(*********************************** G.D S.p.A. - Technical Department ***********************************
============= PROGRAM INFO ============
FOLDER:             TBD
MACHINES INVOLVED:  TBD 

============= DESCRIPTION =============
csp machine declaration

============= REVISIONS ===============
Date		Version	 	Author      	Description             
----------	-------		------------  	--------------------------------------------
2019/04/05 	0000.00	 	M.Grasso		Creation of the PRG
2020/05/05 	0000.01	 	G.Imbriaco		From original author, G.Imbriaco: AccU Change motor with absolute encoder and brake.
										If position_req_mm parameter different from actual_pos_mm and machine reset_edge
										the motor move to position_req then disable again
										Manual movement with basc axis object under test( preset, moving,...)
										All disabled if main accU_Change is not Operational

**********************************************************************************************************)
(*$R process_ref := prc; $*)
PROGRAM csp_case_transport_accU_depth
VAR
	
	prc:											process;
	prc_path:										STRING;
	
	axis:											axis;
	Slot24_drv:										coe_drive;

	not_in_position:								message;
	axis_restore_absolute_position_fb:				restore_absolute_position_with_retain_fb;

	disable_req:									BOOL:=FALSE;
	position_req_mm:								LREAL:=0.0;(*$P unit:= mm; $*)
	move_velocity_req_mms:							LREAL:=10.0;(*$P unit:= mm; $*)
	position_req_tolerance_mm:						LREAL:=0.2;	(*$P $*)
	
	axis_status:									axis_status_enum := AXIS_STATUS_PARAMETERS_START;(*$M $*)
	in_position:									BOOL:=FALSE;(*$M $*)	
	actual_position_mm:								LREAL:=0.0; (*$M unit:= mm; $*)
	axis_move_condition:							BOOL:=FALSE;
	torque_limit:                                   INT := 5000;    (*$P $*)
    torque_limit_old:                               INT;
	
	in_position_motcond:							motorization_conditioner;
	fsm_status:										csp_case_transport_accU_depth_enum;(*$M $*)
	fsm_next_status:								csp_case_transport_accU_depth_enum;
	fsm_enable_condition:							BOOL:=FALSE;
	debug_state_machine:							BOOL:=FALSE;
	debug_state_machine_one_step:					BOOL:=FALSE;
	NC_encoder_val AT %I*:							DINT;
	
END_VAR
VAR PERSISTENT
	per_encoder_val:								UDINT;
	axis_restore_absolute_position_data:			restore_absolute_position_with_retain_struct;
END_VAR

_read_var_input();

_object_manager();

IF NOT objects_running()
THEN
	RETURN;	
END_IF

_read_process_image();

_mode_manager();

CASE process_get_mode(prc) OF
	MODE_ABSENT,
	MODE_INACTIVE:
		RETURN;
	MODE_TEST:
		_handle_process_test();
END_CASE

_set_runtime_properties();

(********************************* BODY *********************************)
//Axis Torque Limit
IF torque_limit <> Torque_limit_old
    THEN
    IF coe_drive_write_parameter(
        index:=16#7010 ,
        complete_access:= FALSE ,
        sub_index:= 16#0B,
        data_source:= ADR(torque_limit),
        data_lenght:= SIZEOF(torque_limit),
        CONVERSION_this:=csp_case_transport_accU_depth.axis.coe_drive^ )= COE_DRIVE_RETURN_VALUE_DONE
       THEN
		 torque_limit_old := Torque_limit;
	END_IF
END_IF

//Axis move condition
IF 	csp_main_accuChange.case_transport_accU_depth_move_req
	OR jog_manager_is_jog_axis_active(SMTR61210_SMTR61200_SMTR61420_CASE_FEED_SHUTTLE_TRANSPORT_AND_DISCHARGE_DEPTH, csp_main_jogManager.jog_manager_accuchange)
THEN
	axis_move_condition := TRUE;
ELSE
	axis_move_condition := FALSE;
END_IF

(*FSM Control*)
fsm_enable_condition := axis_is_ok(FALSE, axis)
						AND
						process_subtree_is_ready(prc)
						AND
						process_get_mode(csp_main_accuChange.prc) = MODE_OPERATIONAL
						AND
						axis_restore_absolute_position_fb.o_position_restored
						AND
						NOT disable_req;		
					
IF	(NOT fsm_enable_condition
	OR
	disable_req)
	AND
	fsm_status <> CSP_CASE_TRANSPORT_ACCU_DEPTH_STATUS_DISABLED
	AND
	fsm_status < CSP_CASE_TRANSPORT_ACCU_DEPTH_STATUS_STOP_REQUEST
THEN
	fsm_status	:=	CSP_CASE_TRANSPORT_ACCU_DEPTH_STATUS_STOP_REQUEST;
END_IF

CASE fsm_status OF
	
	CSP_CASE_TRANSPORT_ACCU_DEPTH_STATUS_NOT_INITIALIZED:
	
        IF	axis_is_ok(return_when_absent := TRUE, CONVERSION_this := axis)
        THEN
            fsm_next_status := CSP_CASE_TRANSPORT_ACCU_DEPTH_STATUS_DISABLED;
        END_IF

		
	CSP_CASE_TRANSPORT_ACCU_DEPTH_STATUS_DISABLED:
	
		IF	fsm_enable_condition
		THEN
			(* Axis with absolute encoder, no home procedure request *)
			fsm_next_status := CSP_CASE_TRANSPORT_ACCU_DEPTH_STATUS_POSITION_CHECK;
		END_IF;
	
		
	CSP_CASE_TRANSPORT_ACCU_DEPTH_STATUS_POSITION_CHECK:

		IF 	axis_move_condition
			OR jog_manager_is_jog_axis_active(SMTR61210_SMTR61200_SMTR61420_CASE_FEED_SHUTTLE_TRANSPORT_AND_DISCHARGE_DEPTH, csp_main_jogManager.jog_manager_accuchange)
		THEN
			fsm_next_status := CSP_CASE_TRANSPORT_ACCU_DEPTH_STATUS_ENABLE_REQUEST;
		END_IF			
	
		
	CSP_CASE_TRANSPORT_ACCU_DEPTH_STATUS_ENABLE_REQUEST:
	
		axis_enable(axis);
		IF axis_is_standstill(axis)
		THEN
			fsm_next_status	:=	CSP_CASE_TRANSPORT_ACCU_DEPTH_STATUS_ENABLED;
		END_IF		

		
	CSP_CASE_TRANSPORT_ACCU_DEPTH_STATUS_ENABLED:
	
		IF 	axis_move_condition
			OR jog_manager_is_jog_axis_active(SMTR61210_SMTR61200_SMTR61420_CASE_FEED_SHUTTLE_TRANSPORT_AND_DISCHARGE_DEPTH, csp_main_jogManager.jog_manager_accuchange)
		THEN
			fsm_next_status	:= CSP_CASE_TRANSPORT_ACCU_DEPTH_STATUS_PHASE_TO_MASTER;	
		END_IF
		
		
	CSP_CASE_TRANSPORT_ACCU_DEPTH_STATUS_PHASE_TO_MASTER:

		IF 	axis.actual_position <> csp_case_transport_accu_virtualMaster.axis.actual_position
			AND ABS(axis.actual_position - csp_case_transport_accu_virtualMaster.axis.actual_position) < 5
		THEN
			axis_move_absolute(
				position 		:= csp_case_transport_accu_virtualMaster.axis.actual_position,
				velocity 		:= move_velocity_req_mms,
				direction		:= AXIS_SHORTEST_WAY,
				acceleration 	:= csp_main_accuChange.CONSTANTS.MAX_ACCELERATION_MMpSEC2 * 0.1,
				deceleration 	:= csp_main_accuChange.CONSTANTS.MAX_DECELERATION_MMpSEC2 * 0.1,
				jerk 			:= csp_main_accuChange.CONSTANTS.MAX_JERK_MMpSEC3, 
				buffer_mode 	:= AXIS_BUFFER_MODE_BUFFERED,
				CONVERSION_this := axis
				); 	
		END_IF
		
		IF 	axis_is_absolute_moving(axis)
			OR axis.actual_position = csp_case_transport_accu_virtualMaster.axis.actual_position
		THEN
			fsm_next_status	:= CSP_CASE_FEED_SHUTTLE_ACCU_DEPTH_STATUS_GEAR_REQUEST;
		END_IF
			
		
	CSP_CASE_TRANSPORT_ACCU_DEPTH_STATUS_GEAR_REQUEST:

		IF	axis_is_standstill(axis)
			AND (
					csp_case_transport_accU_virtualMaster.master_redefined
					OR jog_manager_is_jog_axis_active(SMTR61210_SMTR61200_SMTR61420_CASE_FEED_SHUTTLE_TRANSPORT_AND_DISCHARGE_DEPTH, csp_main_jogManager.jog_manager_accuchange)
				)
		THEN
			axis_engage_position_gear(
				ratio 			:= 1.0,
				acceleration 	:= csp_main_accuChange.CONSTANTS.MAX_ACCELERATION_MMpSEC2 * 0.1,
				deceleration 	:= csp_main_accuChange.CONSTANTS.MAX_DECELERATION_MMpSEC2 * 0.1,
				jerk			:= csp_main_accuChange.CONSTANTS.MAX_JERK_MMpSEC3,
				master 			:= csp_case_transport_accU_virtualMaster.axis,
				CONVERSION_this := axis);
			
		END_IF
		
		IF axis_is_gear_engaging(axis)
		THEN
			fsm_next_status	:=	CSP_CASE_TRANSPORT_ACCU_DEPTH_STATUS_GEARING;
		END_IF

		
	CSP_CASE_TRANSPORT_ACCU_DEPTH_STATUS_GEARING:
		
		IF axis_is_gear_engaged(axis)
		THEN
			fsm_next_status	:=	CSP_CASE_TRANSPORT_ACCU_DEPTH_STATUS_GEARED;
		END_IF
		
		
	CSP_CASE_TRANSPORT_ACCU_DEPTH_STATUS_GEARED:
		
		IF axis_is_moving(csp_case_transport_accU_virtualMaster.axis)
		THEN
			fsm_next_status	:=	CSP_CASE_TRANSPORT_ACCU_DEPTH_STATUS_MOVING;
		END_IF
		
		(* BREAKS GEAR IF NOT JOGGING *)
		IF 	NOT csp_main_accuchange.Brand_Change_Occurred
			AND NOT jog_manager_is_jog_axis_active(SMTR61210_SMTR61200_SMTR61420_CASE_FEED_SHUTTLE_TRANSPORT_AND_DISCHARGE_DEPTH, csp_main_jogManager.jog_manager_accuchange)
		THEN
			fsm_next_status := CSP_CASE_TRANSPORT_ACCU_DEPTH_STATUS_STOP_REQUEST;
		END_IF
		
	
	CSP_CASE_TRANSPORT_ACCU_DEPTH_STATUS_MOVING:

		IF NOT axis_move_condition
			OR ( 
			csp_case_transport_accU_virtualMaster.fsm_status <> CSP_CASE_TRANSPORT_ACCU_VIRTUAL_MASTER_STATUS_ABS_MOVING (* Disables if master disable *)
			AND
			NOT jog_manager_is_jog_axis_active(SMTR61210_SMTR61200_SMTR61420_CASE_FEED_SHUTTLE_TRANSPORT_AND_DISCHARGE_DEPTH, csp_main_jogManager.jog_manager_accuchange)	
				)	
		THEN
			fsm_next_status := CSP_CASE_TRANSPORT_ACCU_DEPTH_STATUS_STOP_REQUEST;
		END_IF
		
		
	CSP_CASE_TRANSPORT_ACCU_DEPTH_STATUS_STOP_REQUEST:

		axis_stop(
		    deceleration 	:= csp_main_accuChange.CONSTANTS.MAX_DECELERATION_MMpSEC2,
		    jerk 			:= csp_main_accuChange.CONSTANTS.MAX_JERK_MMpSEC3,
		    CONVERSION_this 			:= axis);

		IF 	axis_is_standstill(axis)
			OR
			NOT axis_is_ok(FALSE, axis)
			OR
			axis_is_disabled(axis)
		THEN
			fsm_next_status := CSP_CASE_TRANSPORT_ACCU_DEPTH_STATUS_DISABLE_REQUEST;
		END_IF

		
	CSP_CASE_TRANSPORT_ACCU_DEPTH_STATUS_DISABLE_REQUEST:
	
   		axis_disable(axis);
        IF	axis_is_disabled(axis)
        THEN
            fsm_next_status := CSP_CASE_TRANSPORT_ACCU_DEPTH_STATUS_DISABLED;
        END_IF;

END_CASE;

IF NOT debug_state_machine
	OR
	debug_state_machine_one_step
THEN
	fsm_status := fsm_next_status;
	debug_state_machine_one_step := FALSE;
END_IF

(************************************************************************)
_brand_change();

_handle_messages();

_write_output();

ACTION _brand_change:

END_ACTION

ACTION _handle_messages:
IF in_position OR csp_main_jogManager.jog_is_active
THEN
	;//process_message_reset(not_in_position);
ELSE
	IF csp_main_accuChange.machine_size_complete = FALSE
	THEN
		;//process_message_reset(not_in_position);
	ELSE
		;//process_message_set(errorID_1:= 1, errorID_2:= 0, errorID_3:= 0, CONVERSION_this:= not_in_position);
	END_IF
END_IF
END_ACTION

ACTION _handle_process_test:
;
END_ACTION

ACTION _mode_manager:
IF process_mode_req_is_pending(prc)
THEN
    process_apply_mode_req_first_step(prc);
    CASE process_get_mode(prc) OF
        MODE_TO_ABSENT:
			;
        MODE_TO_INACTIVE:
			;
        MODE_TO_TEST:
			;
        MODE_TO_OPERATIONAL:
			;
    END_CASE
    process_apply_mode_req_second_step(prc);
END_IF
END_ACTION

ACTION _object_manager:
IF objects_initialization()
THEN
	sub_process_init(
		object_name						:= 'csp_case_transport_accU_depth.prc', 
		process							:= csp_case_transport_accU.prc, 
		CONVERSION_this					:= prc);
		
	prc_path 							:= process_get_path(prc);
	
	IF csp_main_configurator.Physical_hw 
	THEN
		axis_init(
			object_name					:= CONCAT(prc_path, '_axis'), 
			axis_type					:= AXIS_TYPE_SERVO, 
			encoder_scaling_factor		:= 2.667*0.00000095367431640625, //2.667 mm/rev
			modulo						:= 1024, 
  			process						:= prc, 
			CONVERSION_this				:= axis);
						
		axis_init_absolute_encoder_preset(   
        	position                    := 200, (* 24 COUNT SIZE and Trailing Lugs fit into the guage block width*)
        	CONVERSION_this             := axis);

		axis_add_safety_integrated_series(
			safety_integrated_series	:= csp_case_main_safety_accUChange.sis,
			CONVERSION_this				:= axis);
		axis_set_brake_type(AXIS_BRAKE_DRIVE_CMD, axis);
	ELSE
		axis_init(
			object_name 				:= CONCAT(prc_path, '_axis'),
			axis_type 					:= AXIS_TYPE_VIRTUAL,
			encoder_scaling_factor 		:= G_VIRTUAL_ENCODER_SCALING_FACTOR_DEGPINC,
			modulo 						:= 0,
			process 					:= prc,
			CONVERSION_this 			:= axis);
	END_IF
		
	axis_set_rotation_direction(
		invert_encoder_counting			:= FALSE,
		invert_motor_polarity			:= FALSE,
		CONVERSION_this					:= axis);
		
	coe_drive_init(
		object_name 					:= CONCAT(prc_path, '_Slot24_drv'),
		device_name 					:= 'IO6100Slot24 (EL7211)',
		vendor 							:= DRIVE_BECKHOFF_EL72x1,
		mode 							:= COE_DRIVE_MODE_DRIVEN_BY_AXIS,
		ethercat_master					:= csp_main.cabinet_ethercat_master,
		process							:= prc,
		CONVERSION_this 				:= Slot24_drv);

	axis_add_coe_drive(
		coe_drive						:= Slot24_drv,
		CONVERSION_this					:= axis);
	
	axis_set_max_dynamic(
		reference_velocity				:=	csp_main_accuChange.CONSTANTS.MAX_VELOCITY_MMpSEC,
		velocity						:=	csp_main_accuChange.CONSTANTS.MAX_VELOCITY_MMpSEC,
		acceleration					:=	csp_main_accuChange.CONSTANTS.MAX_ACCELERATION_MMpSEC2,
		deceleration					:=	csp_main_accuChange.CONSTANTS.MAX_DECELERATION_MMpSEC2,
		jerk							:=	csp_main_accuChange.CONSTANTS.MAX_JERK_MMpSEC3,
		following_error					:=	csp_main_accuChange.CONSTANTS.MAX_FOLLOWING_ERROR_MM,
		CONVERSION_this					:=	axis);
	
END_IF

IF objects_running()
THEN
	process_cycle(prc);
	axis_cycle(axis);
	coe_drive_cycle(Slot24_drv);
END_IF
END_ACTION

ACTION _read_process_image:
axis_restore_absolute_position_fb(
	io_retain_data				:= axis_restore_absolute_position_data, 
	io_axis						:= axis);
END_ACTION

ACTION _read_var_input:
;
END_ACTION

ACTION _set_runtime_properties:
axis_status := axis_get_status(axis);
actual_position_mm :=axis_get_actual_modulo_position(axis); (* axis_get_actual_modulo_position(axis); only with modulo*)

IF ABS(position_req_mm - actual_position_mm)< position_req_tolerance_mm
	OR
	process_get_mode(prc)= MODE_ABSENT
	OR
	process_get_mode(csp_main_accuChange.prc) = MODE_ABSENT
THEN
	in_position := TRUE;
ELSE
	in_position := FALSE;	
END_IF
END_ACTION

ACTION _write_output:
;
END_ACTION

END_PROGRAM

(* stored: Version 1.1.0.1, ProductVersion 3.1.4024.3
   POU csp_case_transport_accU_depth: Id {6be1c2f0-ee88-4df3-a979-3915049dda4e}, SpecialFunc None
   Action _brand_change: Id {0995bc08-5e2a-42cb-b2aa-33862f6f74dc}
   Action _handle_messages: Id {515de4c5-676f-499c-ba23-896aa7bc92c5}
   Action _handle_process_test: Id {4a91e919-1ca6-4eae-ac05-9b10b2b711fd}
   Action _mode_manager: Id {2817f95e-bf5a-473e-a2d0-0323239a1e71}
   Action _object_manager: Id {6cadeb71-ae86-4967-88a8-0f9b13cb6454}
   Action _read_process_image: Id {34319212-9b79-410c-8d7d-7a99733d5ea2}
   Action _read_var_input: Id {d3514b9d-5a07-4824-a3f4-017e64de3fa8}
   Action _set_runtime_properties: Id {e5a5edc6-3d70-4c40-87f8-df2f2c949fbd}
   Action _write_output: Id {11302598-bc66-4875-9514-9ee94db5f23d} *)
